FUNCTION_BLOCK FB_Garagepoort
VAR_INPUT
END_VAR
VAR_OUTPUT
END_VAR
VAR
END_VAR

END_FUNCTION_BLOCK

(* stored: Version 1.1.0.1, ProductVersion 3.1.4024.12
   POU FB_Garagepoort: Id {28c07d97-fa80-42dd-841f-b3c5f6f07295}, SpecialFunc None *)
